FUNCTION_BLOCK PAEActFlap EXTENDS PAEActuator1way
VAR_INPUT
END_VAR
VAR_OUTPUT
END_VAR
VAR
END_VAR

METHOD PUBLIC PAEActFlap
VAR_INPUT
END_VAR
END_METHOD

END_FUNCTION_BLOCK

(* stored: Version 1.1.0.1, ProductVersion 3.1.4020.12
   POU PAEActFlap: Id {496459d0-1036-4764-ab4a-0abe57fdc608}, SpecialFunc None
   Method PAEActFlap: Id {fcb52c5d-c9df-4994-aa32-98d559cbdd9d} *)
